FUNCTION_BLOCK Message_Null IMPLEMENTS I_Message
VAR
END_VAR

METHOD Send : HRESULT
VAR_INPUT
	Message	: T_MaxString;
END_VAR
END_METHOD

END_FUNCTION_BLOCK

(* stored: Version 1.1.0.1
   POU Message_Null: Id {9c01881b-903d-4d9c-8c93-cc09793c6e01}, SpecialFunc None
   Method Send: Id {71937b1c-21c1-4a20-b654-041f81015de1} *)
